# EPICS autosave request: iocBoot/ioc2/dbSave/23i_BP_Kb_.req
%
% BURT Request File
%
% 23i:BP:Kb:  BPM @ KB mirrors position
%

file $(DIR)/assy.req ASSY=23i:BP:Kb
file $(DIR)/mtr1.req MTR1=23i:BP:mkb
file $(DIR)/drv1.req DRV1=23i:BP:KBZ
